# EPICS SNL sequencer program: siteApps/seqControls-1.0/seqcontrolsApp/src/gen_SeqControlCV7501.stt
program

option +r;

float groupPVs[43];
assign groupPVs to {
"SCL31-", "SCL31-", "SCL31-",
"SCL31-", "SCL31-", "SCL31-",
"SCL31-", "SCL31-", "SCL31-",
"SCL31-", "SCL31-", "SCL32-",
"SCL32-", "SCL32-", "SCL32-",
"SCL32-", "SCL32-", "SCL32-",
"SCL32-", "SCL32-", "SCL32-",
"SCL32-", "SCL32-", "SCL32-",
"SCL32", "SCL32", "SCL32",
"SCL32", "SCL32", "SCL32",
"SCL32", "SCL32", "SCL32",
"SCL32", "SCL32", "SCL32",
"SCL32", "SCL32", "SCL32",
"SCL32", "SCL32", "SCL32",
"SCL32"
};

float	controlPV;
assign	controlPV to "{C_PV}";
monitor controlPV;
evflag  evControl;
sync 	controlPV evControl;

int index = 0;
int pvcnt = 0;

ss seq_controls_
{
	state init
	{
		when(TRUE)
		{
			efClear(evControl);
		}state WaitEvent
	}

	state WaitEvent
	{
		when(efTestAndClear(evControl))
		{
			index = 0;
			pvcnt = sizeof(groupPVs)/sizeof(groupPVs[0]);
			for(index = 0; index < pvcnt;index++) {
				groupPVs[index] = controlPV;
				pvPut(groupPVs[index], ASYNC);
			}
		}state GrpControls
	}

	state GrpControls
	{
		when(pvArrayPutComplete(groupPVs,TRUE) )
		{
		}state WaitEvent
	}
}
